DEVICE_TYPE FBRT_WINDOW (* An FBRT device showing a window for HMI *)
  (* Standard: 61499 ITA; Description: Copyright (c) 2015 fortiss GmbH This program and the accompanying materials are made available under the terms of the Eclipse Public License 2.0 which is available at https://www.eclipse.org/legal/epl-2.0/ SPDX-License-Identifier: EPL-2.0 *)
  (* Version 1.0, 2015-11-02, Alois Zoitl, fortiss GmbH, Initial version *)
  (* Version 3.0, 2025-04-14, Patrick Aigner, changed package *)
  PACKAGE iec61499::hardware;
  VAR_INPUT
    BOUNDS : ARRAY [0..3] OF DINT; (* Initial[x,y,width,height] *)
    GRID : ARRAY [0..1] OF DINT; (* Grid layout[rows,cols] *)
    MGR_ID : WSTRING := "localhost:61499"; (* Device manager socket ID *)
  END_VAR
END_DEVICE_TYPE
